// TIA Portal V20 export
TYPE "typeCmControlNodeBrakeTest"
// stored: Namespace Unit1.Em4
   STRUCT
      compensator { ExternalWritable := 'False'} : "LER_typeBrakeTestEmControlNodes";
      feedingRoll { S7_SetPoint := 'True'} : "LER_typeBrakeTestEmControlNodes";
      cutter { ExternalWritable := 'False'} : "LER_typeBrakeTestEmControlNodes";
      positionMoving { S7_SetPoint := 'True'} : "LER_typeBrakeTestEmControlNodes";
   END_STRUCT;
END_TYPE
